LIN {X 0,Y 54.036,Z 527.546,A -85,B 0,C 180,E1 -29864.557,E2 -29864.557} C_VEL
LIN {X 0,Y 58.669,Z 527.854,A -85,B 0,C 180,E1 -29873.474,E2 -29873.474} C_VEL
LIN {X 0,Y 64.481,Z 527.558,A -85,B 0,C 180,E1 -29880.96,E2 -29880.96} C_VEL
LIN {X 0,Y 69.082,Z 526.912,A -85,B 0,C 180,E1 -29884.107,E2 -29884.107} C_VEL
LIN {X 0,Y 78.027,Z 525.099,A -85,B 0,C 180,E1 -29887.878,E2 -29887.878} C_VEL
LIN {X 0,Y 83.488,Z 523.571,A -85,B 0,C 180,E1 -29889.694,E2 -29889.694} C_VEL
LIN {X 0,Y 84.39,Z 523.544,A -85,B 0,C 180,E1 -29894.47,E2 -29894.47} C_VEL
LIN {X 0,Y 84.222,Z 523.754,A -85,B 0,C 180,E1 -29896.308,E2 -29896.308} C_VEL
LIN {X 0,Y 83.259,Z 524.243,A -85,B 0,C 180,E1 -29898.269,E2 -29898.269} C_VEL
LIN {X 0,Y 75.2,Z 526.708,A -85,B 0,C 180,E1 -29900.878,E2 -29900.878} C_VEL
LIN {X 0,Y 62.904,Z 529.265,A -85,B 0,C 180,E1 -29906.679,E2 -29906.679} C_VEL
LIN {X 0,Y 51.648,Z 530.299,A -85,B 0,C 180,E1 -29915.3,E2 -29915.3} C_VEL
LIN {X 0,Y 42.225,Z 529.751,A -85,B 0,C 180,E1 -29928.288,E2 -29928.288} C_VEL
LIN {X 0,Y 38.734,Z 528.937,A -85,B 0,C 180,E1 -29937.05,E2 -29937.05} C_VEL
LIN {X 0,Y 36.311,Z 527.697,A -85,B 0,C 180,E1 -29947.253,E2 -29947.253} C_VEL
LIN {X 0,Y 35.574,Z 523.998,A -85,B 0,C 180,E1 -29970.025,E2 -29970.025} C_VEL
LIN {X 0,Y 36.876,Z 521.96,A -85,B 0,C 180,E1 -29979.624,E2 -29979.624} C_VEL
LIN {X 0,Y 38.775,Z 527.432,A -85,B 0,C 180,E1 -29996.389,E2 -29996.389} C_VEL
LIN {X 0,Y 45.345,Z 533.082,A -85,B 0,C 180,E1 -30014.249,E2 -30014.249} C_VEL
LIN {X 0,Y 52.383,Z 536.251,A -85,B 0,C 180,E1 -30023.637,E2 -30023.637} C_VEL
LIN {X 0,Y 59.68,Z 538.549,A -85,B 0,C 180,E1 -30029.758,E2 -30029.758} C_VEL
LIN {X 0,Y 60.796,Z 538.755,A -85,B 0,C 180,E1 -30032.455,E2 -30032.455} C_VEL
LIN {X 0,Y 52.766,Z 535.916,A -85,B 0,C 180,E1 -30038.846,E2 -30038.846} C_VEL
LIN {X 0,Y 43.689,Z 531.082,A -85,B 0,C 180,E1 -30050.74,E2 -30050.74} C_VEL
LIN {X 0,Y 37.979,Z 525.719,A -85,B 0,C 180,E1 -30065.305,E2 -30065.305} C_VEL
LIN {X 0,Y 35.275,Z 518.979,A -85,B 0,C 180,E1 -30083.478,E2 -30083.478} C_VEL
LIN {X 0,Y 35.443,Z 513.027,A -85,B 0,C 180,E1 -30097.478,E2 -30097.478} C_VEL
LIN {X 0,Y 37.45,Z 504.518,A -85,B 0,C 180,E1 -30113.136,E2 -30113.136} C_VEL
LIN {X 0,Y 40.393,Z 496.567,A -85,B 0,C 180,E1 -30123.777,E2 -30123.777} C_VEL
LIN {X 0,Y 41.813,Z 497.334,A -85,B 0,C 180,E1 -30127.577,E2 -30127.577} C_VEL
LIN {X 0,Y 44.62,Z 497.247,A -85,B 0,C 180,E1 -30130.908,E2 -30130.908} C_VEL
LIN {X 0,Y 46.366,Z 496.981,A -85,B 0,C 180,E1 -30132.333,E2 -30132.333} C_VEL
LIN {X 0,Y 47.983,Z 497.364,A -85,B 0,C 180,E1 -30134.62,E2 -30134.62} C_VEL
LIN {X 0,Y 47.031,Z 499.316,A -85,B 0,C 180,E1 -30137.028,E2 -30137.028} C_VEL
LIN {X 0,Y 41.347,Z 506.796,A -85,B 0,C 180,E1 -30147.044,E2 -30147.044} C_VEL
LIN {X 0,Y 36.726,Z 513.38,A -85,B 0,C 180,E1 -30161.007,E2 -30161.007} C_VEL
LIN {X 0,Y 34.405,Z 518.941,A -85,B 0,C 180,E1 -30179.425,E2 -30179.425} C_VEL
LIN {X 0,Y 36.135,Z 523.579,A -85,B 0,C 180,E1 -30201.035,E2 -30201.035} C_VEL
LIN {X 0,Y 39.49,Z 525.629,A -85,B 0,C 180,E1 -30212.8,E2 -30212.8} C_VEL
LIN {X 0,Y 45.361,Z 527.218,A -85,B 0,C 180,E1 -30224.186,E2 -30224.186} C_VEL
LIN {X 0,Y 51.969,Z 527.997,A -85,B 0,C 180,E1 -30232.231,E2 -30232.231} C_VEL
LIN {X 0,Y 61.733,Z 527.845,A -85,B 0,C 180,E1 -30240.002,E2 -30240.002} C_VEL
LIN {X 0,Y 69.082,Z 526.912,A -85,B 0,C 180,E1 -30244.107,E2 -30244.107} C_VEL
LIN {X 0,Y 69.967,Z 526.835,A -85,B 0,C 180,E1 -30245.229,E2 -30245.229} C_VEL
LIN {X 0,Y 69.844,Z 526.982,A -85,B 0,C 180,E1 -30247.595,E2 -30247.595} C_VEL
LIN {X 0,Y 67.75,Z 527.505,A -85,B 0,C 180,E1 -30251.156,E2 -30251.156} C_VEL
LIN {X 0,Y 65.475,Z 527.951,A -85,B 0,C 180,E1 -30253.59,E2 -30253.59} C_VEL
LIN {X 0,Y 60.018,Z 528.926,A -85,B 0,C 180,E1 -30258.401,E2 -30258.401} C_VEL
LIN {X 0,Y 53.256,Z 529.677,A -85,B 0,C 180,E1 -30264.155,E2 -30264.155} C_VEL
LIN {X 0,Y 50.147,Z 529.771,A -85,B 0,C 180,E1 -30266.558,E2 -30266.558} C_VEL
LIN {X 0,Y 42.297,Z 529.669,A -85,B 0,C 180,E1 -30273.861,E2 -30273.861} C_VEL
LIN {X 0,Y 37.215,Z 529.116,A -85,B 0,C 180,E1 -30280.978,E2 -30280.978} C_VEL
LIN {X 0,Y 29.901,Z 526.809,A -85,B 0,C 180,E1 -30301.995,E2 -30301.995} C_VEL
LIN {X 0,Y 28.258,Z 523.837,A -85,B 0,C 180,E1 -30324.22,E2 -30324.22} C_VEL
LIN {X 0,Y 30.399,Z 520.266,A -85,B 0,C 180,E1 -30343.707,E2 -30343.707} C_VEL
LIN {X 0,Y 33.378,Z 526.111,A -85,B 0,C 180,E1 -30363.937,E2 -30363.937} C_VEL
LIN {X 0,Y 40.69,Z 531.394,A -85,B 0,C 180,E1 -30381.041,E2 -30381.041} C_VEL
LIN {X 0,Y 48.589,Z 534.85,A -85,B 0,C 180,E1 -30390.245,E2 -30390.245} C_VEL
LIN {X 0,Y 47.34,Z 534.247,A -85,B 0,C 180,E1 -30393.549,E2 -30393.549} C_VEL
LIN {X 0,Y 38.609,Z 529.648,A -85,B 0,C 180,E1 -30404.151,E2 -30404.151} C_VEL
LIN {X 0,Y 31.087,Z 522.898,A -85,B 0,C 180,E1 -30423.236,E2 -30423.236} C_VEL
LIN {X 0,Y 28.384,Z 515.584,A -85,B 0,C 180,E1 -30445.668,E2 -30445.668} C_VEL
LIN {X 0,Y 28.966,Z 508.843,A -85,B 0,C 180,E1 -30463.247,E2 -30463.247} C_VEL
LIN {X 0,Y 31.333,Z 501.145,A -85,B 0,C 180,E1 -30478.767,E2 -30478.767} C_VEL
LIN {X 0,Y 31.874,Z 501.675,A -85,B 0,C 180,E1 -30481.871,E2 -30481.871} C_VEL
LIN {X 0,Y 32.828,Z 501.912,A -85,B 0,C 180,E1 -30484.619,E2 -30484.619} C_VEL
LIN {X 0,Y 37.064,Z 501.89,A -85,B 0,C 180,E1 -30491.445,E2 -30491.445} C_VEL
LIN {X 0,Y 38.475,Z 502.916,A -85,B 0,C 180,E1 -30495.671,E2 -30495.671} C_VEL
LIN {X 0,Y 31.982,Z 510.585,A -85,B 0,C 180,E1 -30509.972,E2 -30509.972} C_VEL
LIN {X 0,Y 28.136,Z 516.285,A -85,B 0,C 180,E1 -30528.16,E2 -30528.16} C_VEL
LIN {X 0,Y 27.462,Z 520.809,A -85,B 0,C 180,E1 -30549.856,E2 -30549.856} C_VEL
LIN {X 0,Y 31.605,Z 524.824,A -85,B 0,C 180,E1 -30573.598,E2 -30573.598} C_VEL
LIN {X 0,Y 39.501,Z 527.318,A -85,B 0,C 180,E1 -30589.755,E2 -30589.755} C_VEL
LIN {X 0,Y 49.219,Z 528.434,A -85,B 0,C 180,E1 -30600.003,E2 -30600.003} C_VEL
LIN {X 0,Y 59.915,Z 528.29,A -85,B 0,C 180,E1 -30606.739,E2 -30606.739} C_VEL
LIN {X 0,Y 71.726,Z 526.72,A -85,B 0,C 180,E1 -30611.592,E2 -30611.592} C_VEL
LIN {X 0,Y 76.119,Z 525.806,A -85,B 0,C 180,E1 -30612.948,E2 -30612.948} C_VEL
LIN {X 0,Y 77.312,Z 525.548,A -85,B 0,C 180,E1 -30613.689,E2 -30613.689} C_VEL
LIN {X 0,Y 74.818,Z 526.285,A -85,B 0,C 180,E1 -30615.135,E2 -30615.135} C_VEL
LIN {X 0,Y 66.435,Z 528.087,A -85,B 0,C 180,E1 -30617.857,E2 -30617.857} C_VEL
LIN {X 0,Y 60.046,Z 529.075,A -85,B 0,C 180,E1 -30620.599,E2 -30620.599} C_VEL
LIN {X 0,Y 50.147,Z 529.771,A -85,B 0,C 180,E1 -30626.558,E2 -30626.558} C_VEL
LIN {X 0,Y 44.934,Z 529.781,A -85,B 0,C 180,E1 -30629.935,E2 -30629.935} C_VEL
LIN {X 0,Y 35.804,Z 528.926,A -85,B 0,C 180,E1 -30635.385,E2 -30635.385} C_VEL
LIN {X 0,Y 27.381,Z 527.246,A -85,B 0,C 180,E1 -30644.421,E2 -30644.421} C_VEL
LIN {X 0,Y 23.784,Z 525.858,A -85,B 0,C 180,E1 -30654.455,E2 -30654.455} C_VEL
LIN {X 0,Y 21.525,Z 521.73,A -85,B 0,C 180,E1 -30690.042,E2 -30690.042} C_VEL
LIN {X 0,Y 24.158,Z 518.492,A -85,B 0,C 180,E1 -30710.147,E2 -30710.147} C_VEL
LIN {X 0,Y 27.573,Z 523.562,A -85,B 0,C 180,E1 -30730.115,E2 -30730.115} C_VEL
LIN {X 0,Y 35.707,Z 529.045,A -85,B 0,C 180,E1 -30747.991,E2 -30747.991} C_VEL
LIN {X 0,Y 37.473,Z 529.902,A -85,B 0,C 180,E1 -30751.651,E2 -30751.651} C_VEL
LIN {X 0,Y 27.42,Z 523.159,A -85,B 0,C 180,E1 -30768.912,E2 -30768.912} C_VEL
LIN {X 0,Y 22.011,Z 515.238,A -85,B 0,C 180,E1 -30796.547,E2 -30796.547} C_VEL
LIN {X 0,Y 21.815,Z 508.48,A -85,B 0,C 180,E1 -30820.106,E2 -30820.106} C_VEL
LIN {X 0,Y 22.558,Z 505.282,A -85,B 0,C 180,E1 -30829.642,E2 -30829.642} C_VEL
LIN {X 0,Y 24.267,Z 506.002,A -85,B 0,C 180,E1 -30840.313,E2 -30840.313} C_VEL
LIN {X 0,Y 29.417,Z 506.282,A -85,B 0,C 180,E1 -30852.851,E2 -30852.851} C_VEL
LIN {X 0,Y 28.709,Z 507.415,A -85,B 0,C 180,E1 -30855.798,E2 -30855.798} C_VEL
LIN {X 0,Y 22.548,Z 514.135,A -85,B 0,C 180,E1 -30875.672,E2 -30875.672} C_VEL
LIN {X 0,Y 20.174,Z 518.942,A -85,B 0,C 180,E1 -30901.452,E2 -30901.452} C_VEL
LIN {X 0,Y 23.493,Z 523.56,A -85,B 0,C 180,E1 -30933.737,E2 -30933.737} C_VEL
LIN {X 0,Y 28.663,Z 525.841,A -85,B 0,C 180,E1 -30948.584,E2 -30948.584} C_VEL
LIN {X 0,Y 36.652,Z 527.752,A -85,B 0,C 180,E1 -30960.004,E2 -30960.004} C_VEL
LIN {X 0,Y 47.472,Z 528.872,A -85,B 0,C 180,E1 -30968.517,E2 -30968.517} C_VEL
LIN {X 0,Y 57.766,Z 528.796,A -85,B 0,C 180,E1 -30973.34,E2 -30973.34} C_VEL
LIN {X 0,Y 57.924,Z 528.822,A -85,B 0,C 180,E1 -30973.987,E2 -30973.987} C_VEL
LIN {X 0,Y 44.942,Z 529.385,A -85,B 0,C 180,E1 -30980.296,E2 -30980.296} C_VEL
LIN {X 0,Y 38.79,Z 529.095,A -85,B 0,C 180,E1 -30985.114,E2 -30985.114} C_VEL
LIN {X 0,Y 27.904,Z 527.354,A -85,B 0,C 180,E1 -31000.974,E2 -31000.974} C_VEL
LIN {X 0,Y 23.784,Z 525.858,A -85,B 0,C 180,E1 -31014.455,E2 -31014.455} C_VEL
LIN {X 0,Y 21.724,Z 524.795,A -85,B 0,C 180,E1 -31022.523,E2 -31022.523} C_VEL
LIN {X 0,Y 17.843,Z 522.548,A -85,B 0,C 180,E1 -31037.147,E2 -31037.147} C_VEL
LIN {X 0,Y 15.602,Z 519.884,A -85,B 0,C 180,E1 -31057.292,E2 -31057.292} C_VEL
LIN {X 0,Y 16.355,Z 518.21,A -85,B 0,C 180,E1 -31070.16,E2 -31070.16} C_VEL
LIN {X 0,Y 18.425,Z 516.591,A -85,B 0,C 180,E1 -31080.511,E2 -31080.511} C_VEL
LIN {X 0,Y 25.176,Z 522.926,A -85,B 0,C 180,E1 -31106.936,E2 -31106.936} C_VEL
LIN {X 0,Y 26.545,Z 523.773,A -85,B 0,C 180,E1 -31110.567,E2 -31110.567} C_VEL
LIN {X 0,Y 17.701,Z 516.347,A -85,B 0,C 180,E1 -31134.296,E2 -31134.296} C_VEL
LIN {X 0,Y 14.799,Z 509.157,A -85,B 0,C 180,E1 -31168.343,E2 -31168.343} C_VEL
LIN {X 0,Y 19.376,Z 510.027,A -85,B 0,C 180,E1 -31208.684,E2 -31208.684} C_VEL
LIN {X 0,Y 19.416,Z 510.904,A -85,B 0,C 180,E1 -31214.201,E2 -31214.201} C_VEL
LIN {X 0,Y 13.483,Z 517.261,A -85,B 0,C 180,E1 -31249.278,E2 -31249.278} C_VEL
LIN {X 0,Y 15.479,Z 522.068,A -85,B 0,C 180,E1 -31295.099,E2 -31295.099} C_VEL
LIN {X 0,Y 23.81,Z 525.679,A -85,B 0,C 180,E1 -31320.006,E2 -31320.006} C_VEL
LIN {X 0,Y 35.922,Z 528.292,A -85,B 0,C 180,E1 -31332.102,E2 -31332.102} C_VEL
LIN {X 0,Y 36.349,Z 528.457,A -85,B 0,C 180,E1 -31334.923,E2 -31334.923} C_VEL
LIN {X 0,Y 29.888,Z 527.67,A -85,B 0,C 180,E1 -31339.945,E2 -31339.945} C_VEL
LIN {X 0,Y 23.862,Z 526.505,A -85,B 0,C 180,E1 -31348.004,E2 -31348.004} C_VEL
LIN {X 0,Y 15.093,Z 522.955,A -85,B 0,C 180,E1 -31382.315,E2 -31382.315} C_VEL
LIN {X 0,Y 15.455,Z 519.134,A -85,B 0,C 180,E1 -31423.201,E2 -31423.201} C_VEL
LIN {X 0,Y 16.355,Z 518.21,A -85,B 0,C 180,E1 -31430.16,E2 -31430.16} C_VEL
LIN {X 0,Y 16.518,Z 517.344,A -85,B 0,C 180,E1 -31436.101,E2 -31436.101} C_VEL
LIN {X 0,Y 15.567,Z 516.268,A -85,B 0,C 180,E1 -31443.981,E2 -31443.981} C_VEL
LIN {X 0,Y 13.31,Z 515.026,A -85,B 0,C 180,E1 -31456.102,E2 -31456.102} C_VEL
LIN {X 0,Y 10.428,Z 514.135,A -85,B 0,C 180,E1 -31473.801,E2 -31473.801} C_VEL
LIN {X 0,Y 8.337,Z 513.33,A -85,B 0,C 180,E1 -31513.93,E2 -31513.93} C_VEL
LIN {X 0,Y 8.878,Z 513.108,A -85,B 0,C 180,E1 -31536.34,E2 -31536.34} C_VEL
LIN {X 0,Y 10.946,Z 513.335,A -85,B 0,C 180,E1 -31564.227,E2 -31564.227} C_VEL
LIN {X 0,Y 7.03,Z 516.494,A -85,B 0,C 180,E1 -31591.965,E2 -31591.965} C_VEL
LIN {X 0,Y 11.044,Z 522.156,A -85,B 0,C 180,E1 -31680.012,E2 -31680.012} C_VEL
LIN {X 0,Y 16.858,Z 524.352,A -85,B 0,C 180,E1 -31692.237,E2 -31692.237} C_VEL
LIN {X 0,Y 14.963,Z 523.907,A -85,B 0,C 180,E1 -31700.232,E2 -31700.232} C_VEL
LIN {X 0,Y 7.568,Z 520.341,A -85,B 0,C 180,E1 -31748.273,E2 -31748.273} C_VEL
LIN {X 0,Y 12.5,Z 515.355,A -85,B 0,C 180,E1 -31814.753,E2 -31814.753} C_VEL
LIN {X 0,Y 13.937,Z 514.607,A -85,B 0,C 180,E1 -31819.243,E2 -31819.243} C_VEL
LIN {X 0,Y 14.888,Z 515.506,A -85,B 0,C 180,E1 -31824.276,E2 -31824.276} C_VEL
LIN {X 0,Y 14.553,Z 515.266,A -85,B 0,C 180,E1 -31831.113,E2 -31831.113} C_VEL
LIN {X 0,Y 11.907,Z 512.927,A -85,B 0,C 180,E1 -31840.598,E2 -31840.598} C_VEL
LIN {X 0,Y 8.828,Z 513.376,A -85,B 0,C 180,E1 -31859.984,E2 -31859.984} C_VEL
LIN {X 0,Y 8.878,Z 513.108,A -85,B 0,C 180,E1 -31896.34,E2 -31896.34} C_VEL
LIN {X 0,Y 9.754,Z 515.105,A -85,B 0,C 180,E1 -31908.093,E2 -31908.093} C_VEL
LIN {X 0,Y 9.754,Z 600,A -85,B 0,C 180,E1 -31908.093,E2 -31908.093} C_VEL
LIN {X 0,Y 9.754,Z 600,A -85,B 0,C 180,E1 -31908.093,E2 -31908.093}

QRS_NEXT_CUT()

QRS_NEXT()
QRS_HOME()

END
